// TIA Portal V20 export
TYPE "typeCmControlNodeSoftCamthicknessAxisZ"
// stored: Namespace Unit1.Em8
   STRUCT
      pos00_wait : "LER_typeSoftCamPosition";
      pos01_workReady : "LER_typeSoftCamPosition";
      pos02_thickness : "LER_typeSoftCamPosition";
      pos03_position : "LER_typeSoftCamPosition";
      pos04_position : "LER_typeSoftCamPosition";
      pos05_position : "LER_typeSoftCamPosition";
      pos06_position : "LER_typeSoftCamPosition";
      pos07_position : "LER_typeSoftCamPosition";
      pos08_position : "LER_typeSoftCamPosition";
      pos09_position : "LER_typeSoftCamPosition";
      pos10_position : "LER_typeSoftCamPosition";
      pos11_position : "LER_typeSoftCamPosition";
      pos12_position : "LER_typeSoftCamPosition";
      pos13_position : "LER_typeSoftCamPosition";
      pos14_position : "LER_typeSoftCamPosition";
      pos15_position : "LER_typeSoftCamPosition";
   END_STRUCT;
END_TYPE
